// SIMATIC S7-200 project (STEP 7-Micro/WIN), CPU 221 REL 01.10

ORGANIZATION_BLOCK 主程序:OB1
TITLE=程序注释
BEGIN
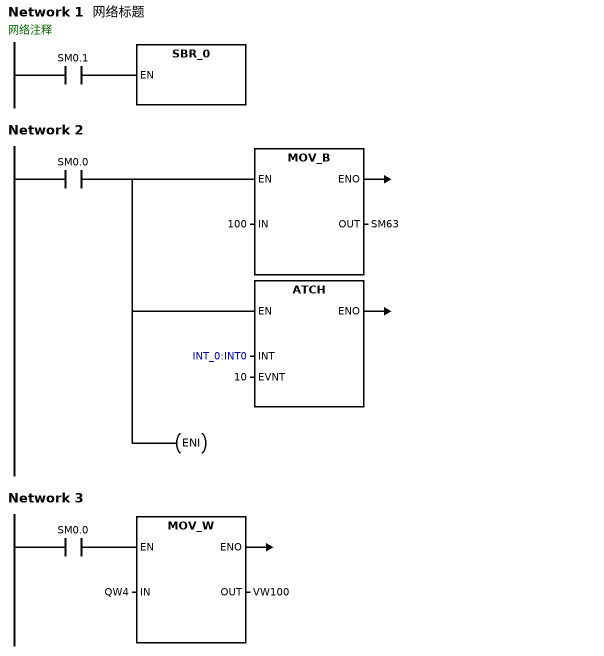
Network 1 // 网络标题
// 网络注释
LD     SM0.1
CALL   SBR_0:SBR0
Network 2
// (network saved uncompiled; LAD cells follow)
// row 0: c0 -| |- SM0.0 v  c1 --  c2 [MOV_B EN:=power@row0, IN:=100, ENO=>power, OUT=>SM63]  c3 ->
// row 1: c0 ^v  c2 [box]
// row 2: c0 ^v  c1 --  c2 [ATCH EN:=power@row2, INT:=INT_0:INT0, EVNT:=10, ENO=>power]  c3 ->
// row 3: c0 ^v  c2 [box]
// row 4: c0 ^  c1 -(ENI)
Network 3
LD     SM0.0
MOVW   QW4, VW100
END_ORGANIZATION_BLOCK
